// SIMATIC S7-200 project (STEP 7-Micro/WIN), CPU 226 CN REL 02.01

ORGANIZATION_BLOCK MAIN:OB1
TITLE=PROGRAM COMMENTS
BEGIN
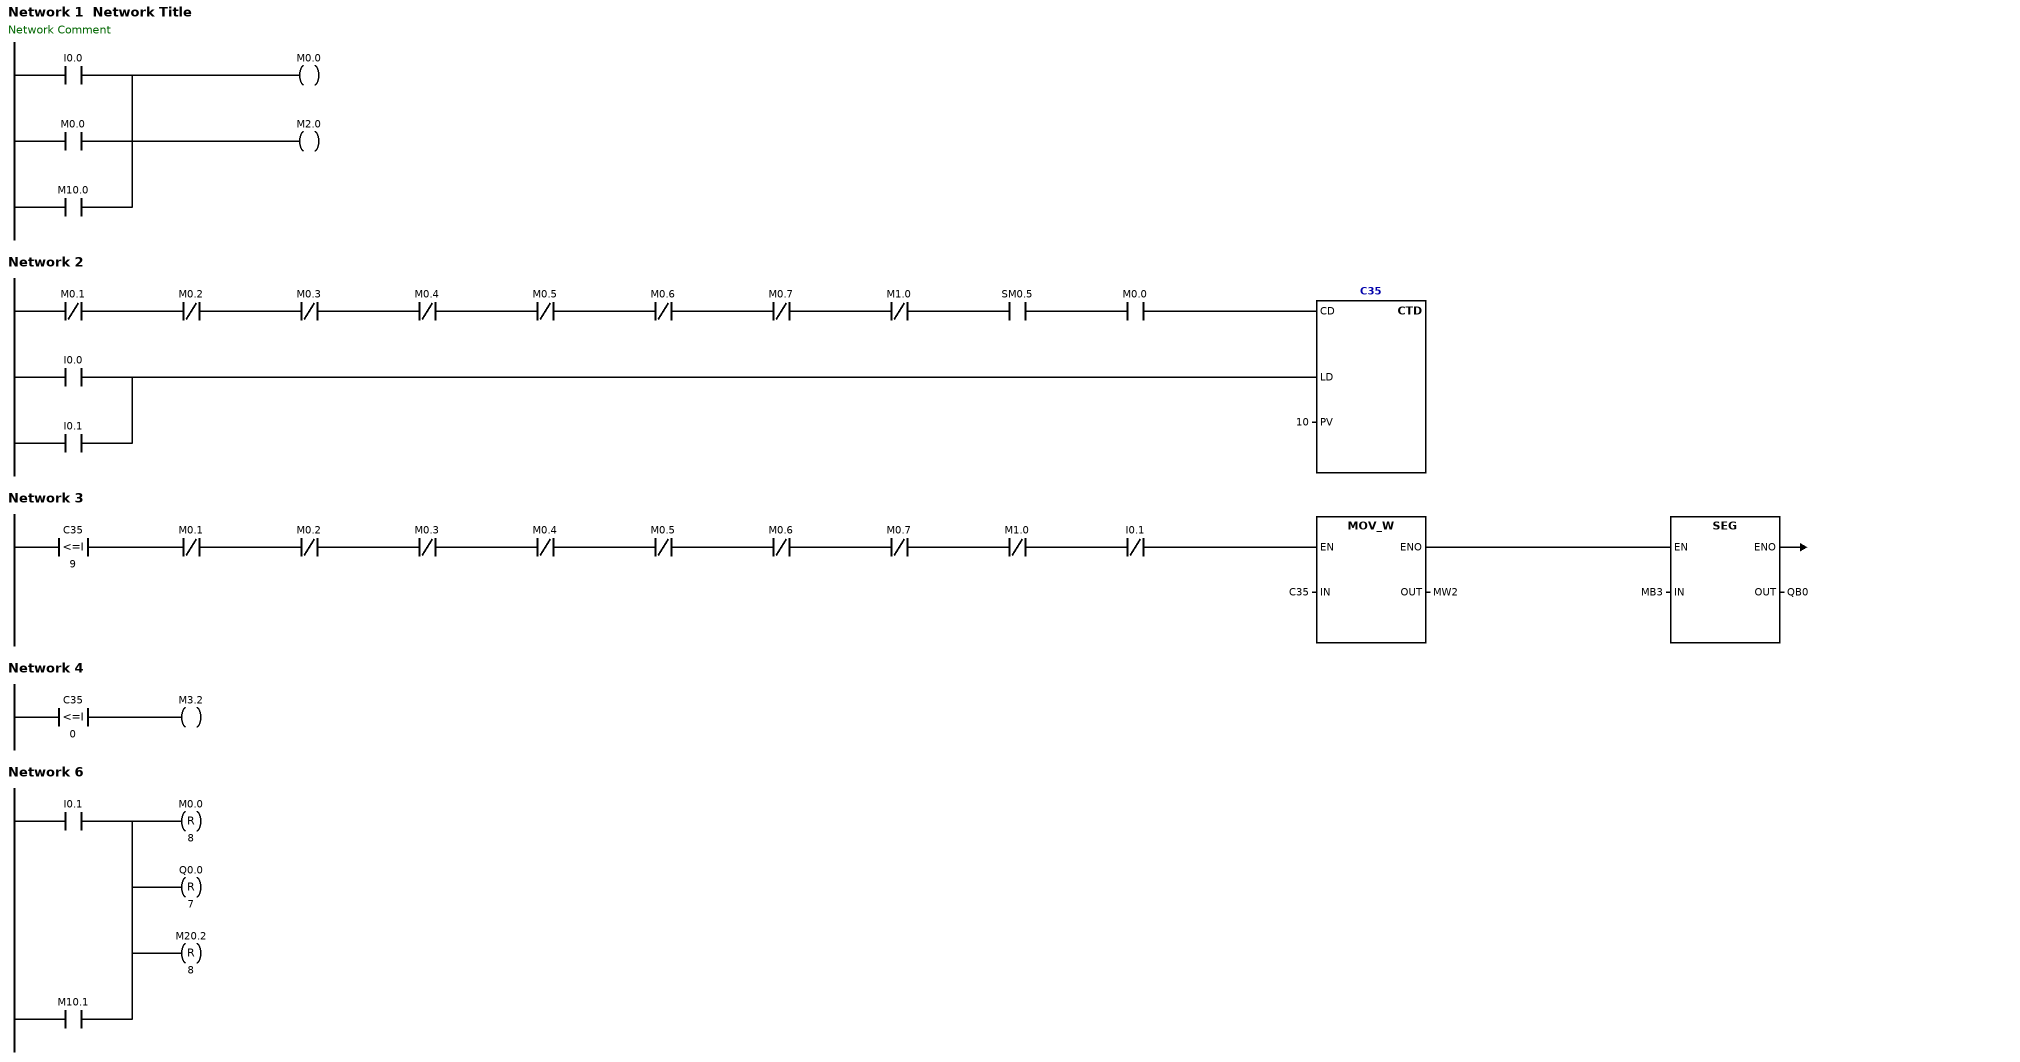
Network 1 // Network Title
// Network Comment
// (network saved uncompiled; LAD cells follow)
// row 0: c0 -| |- I0.0 v  c1 --  c2 -( ) M0.0
// row 1: c0 -| |- M0.0 ^v  c1 --  c2 -( ) M2.0
// row 2: c0 -| |- M10.0 ^
Network 2
LDN    M0.1
AN     M0.2
AN     M0.3
AN     M0.4
AN     M0.5
AN     M0.6
AN     M0.7
AN     M1.0
A      SM0.5
A      M0.0
LD     I0.0
O      I0.1
CTD    C35, 10
Network 3
LDW<=  C35, 9
AN     M0.1
AN     M0.2
AN     M0.3
AN     M0.4
AN     M0.5
AN     M0.6
AN     M0.7
AN     M1.0
AN     I0.1
MOVW   C35, MW2
AENO
SEG    MB3, QB0
Network 4
LDW<=  C35, 0
=      M3.2
Network 6
// (network saved uncompiled; LAD cells follow)
// row 0: c0 -| |- I0.1 v  c1 -(R) M0.0, 8
// row 1: c0 ^v  c1 -(R) Q0.0, 7
// row 2: c0 ^v  c1 -(R) M20.2, 8
// row 3: c0 -| |- M10.1 ^
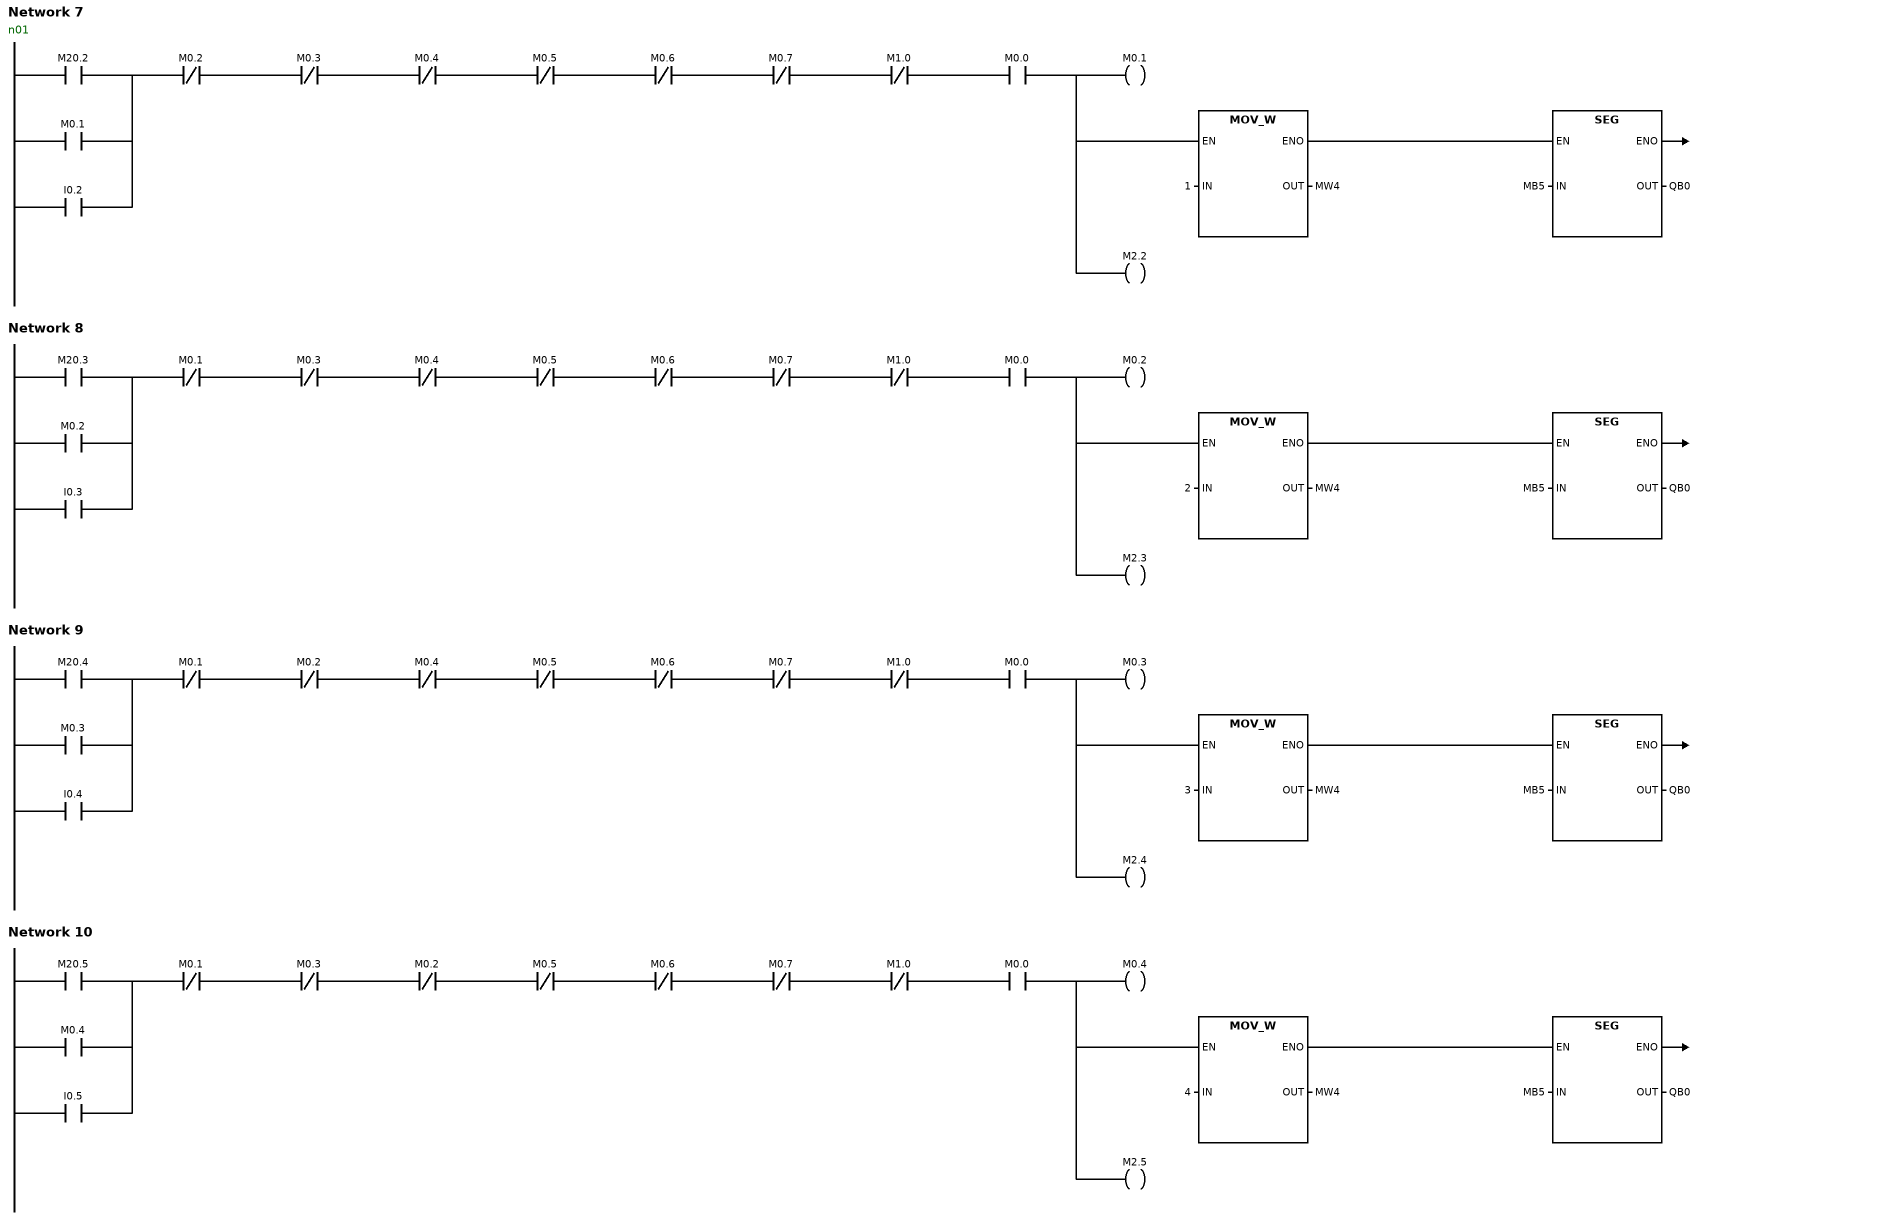
Network 7
// n01
LD     M20.2
O      M0.1
O      I0.2
AN     M0.2
AN     M0.3
AN     M0.4
AN     M0.5
AN     M0.6
AN     M0.7
AN     M1.0
A      M0.0
LPS
=      M0.1
MOVW   1, MW4
AENO
SEG    MB5, QB0
LPP
=      M2.2
Network 8
LD     M20.3
O      M0.2
O      I0.3
AN     M0.1
AN     M0.3
AN     M0.4
AN     M0.5
AN     M0.6
AN     M0.7
AN     M1.0
A      M0.0
LPS
=      M0.2
MOVW   2, MW4
AENO
SEG    MB5, QB0
LPP
=      M2.3
Network 9
LD     M20.4
O      M0.3
O      I0.4
AN     M0.1
AN     M0.2
AN     M0.4
AN     M0.5
AN     M0.6
AN     M0.7
AN     M1.0
A      M0.0
LPS
=      M0.3
MOVW   3, MW4
AENO
SEG    MB5, QB0
LPP
=      M2.4
Network 10
LD     M20.5
O      M0.4
O      I0.5
AN     M0.1
AN     M0.3
AN     M0.2
AN     M0.5
AN     M0.6
AN     M0.7
AN     M1.0
A      M0.0
LPS
=      M0.4
MOVW   4, MW4
AENO
SEG    MB5, QB0
LPP
=      M2.5
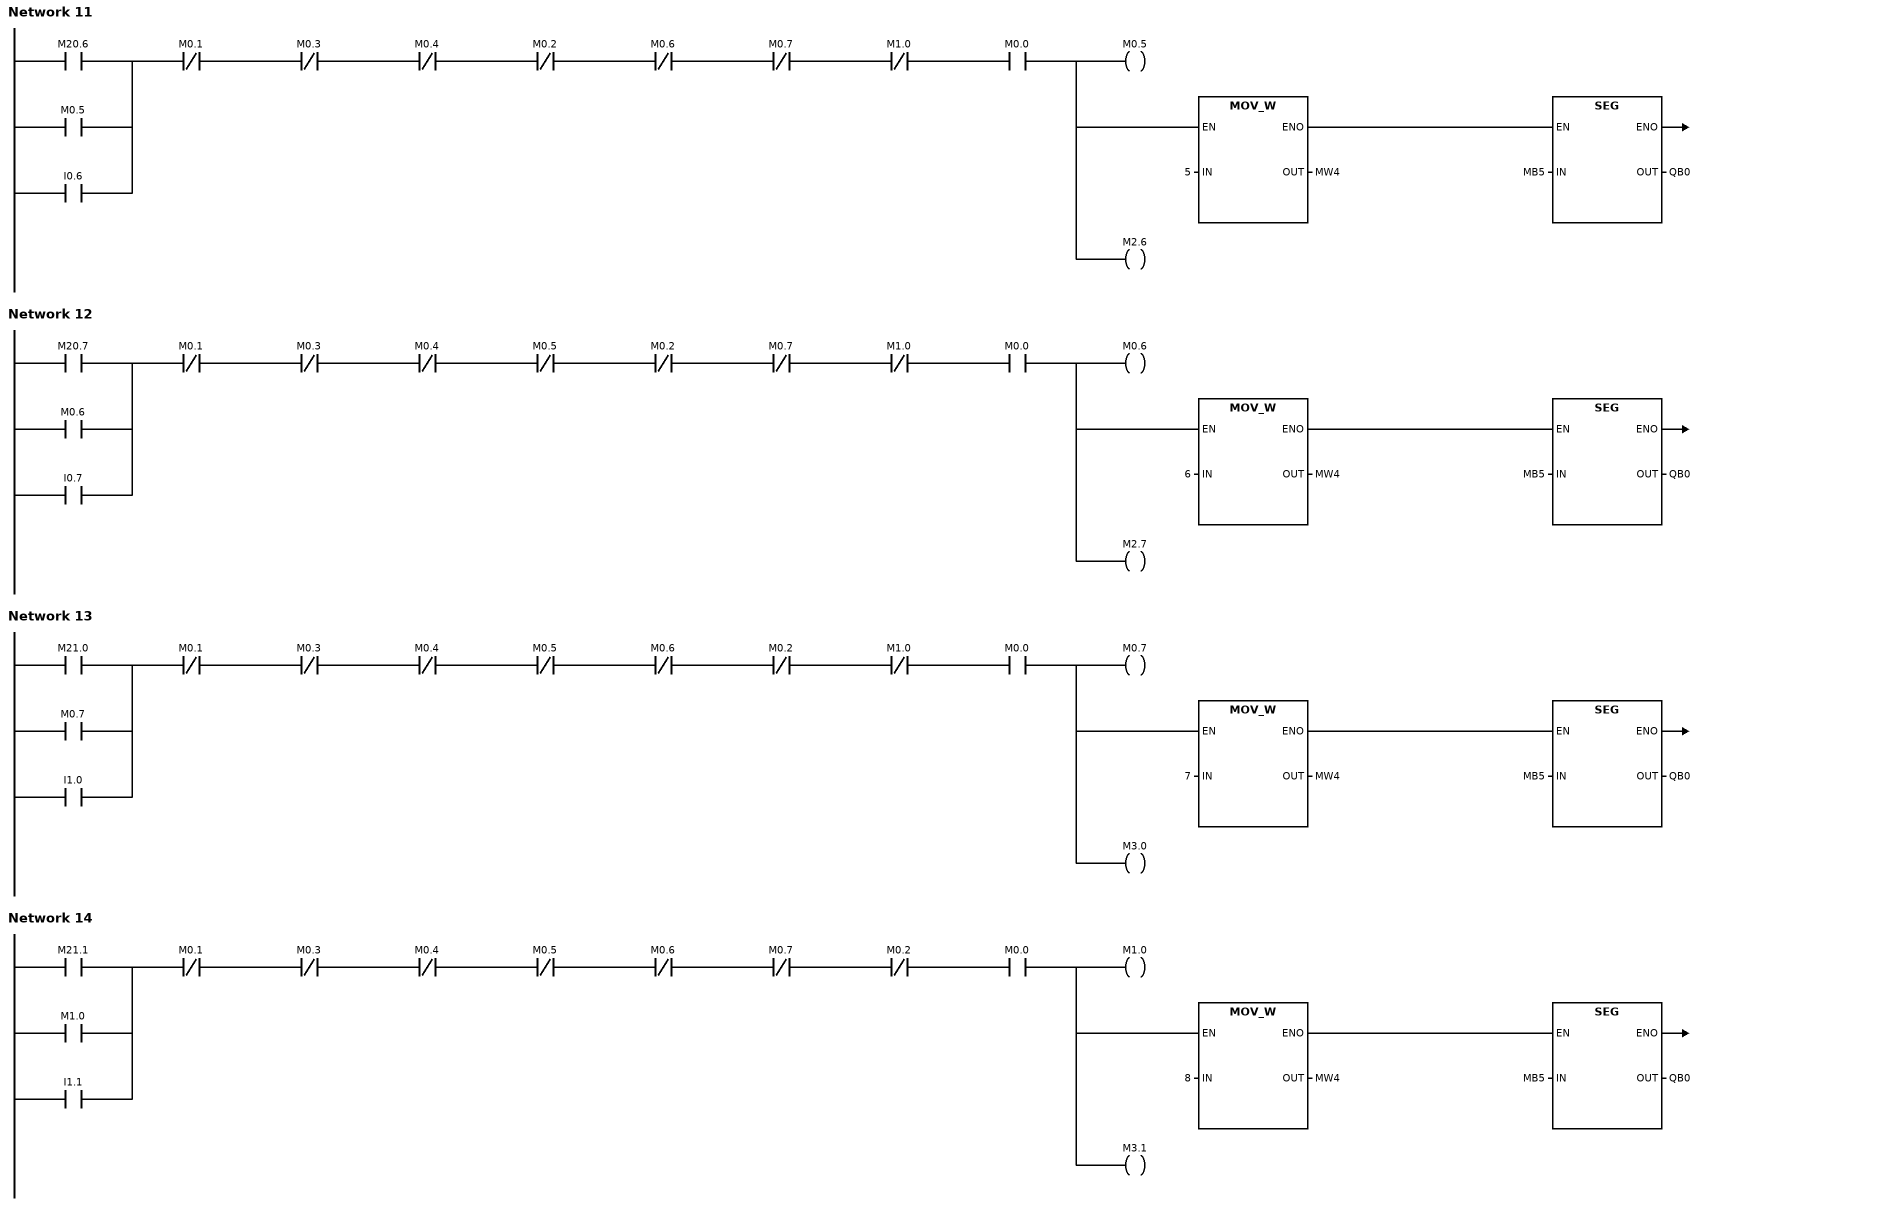
Network 11
LD     M20.6
O      M0.5
O      I0.6
AN     M0.1
AN     M0.3
AN     M0.4
AN     M0.2
AN     M0.6
AN     M0.7
AN     M1.0
A      M0.0
LPS
=      M0.5
MOVW   5, MW4
AENO
SEG    MB5, QB0
LPP
=      M2.6
Network 12
LD     M20.7
O      M0.6
O      I0.7
AN     M0.1
AN     M0.3
AN     M0.4
AN     M0.5
AN     M0.2
AN     M0.7
AN     M1.0
A      M0.0
LPS
=      M0.6
MOVW   6, MW4
AENO
SEG    MB5, QB0
LPP
=      M2.7
Network 13
LD     M21.0
O      M0.7
O      I1.0
AN     M0.1
AN     M0.3
AN     M0.4
AN     M0.5
AN     M0.6
AN     M0.2
AN     M1.0
A      M0.0
LPS
=      M0.7
MOVW   7, MW4
AENO
SEG    MB5, QB0
LPP
=      M3.0
Network 14
LD     M21.1
O      M1.0
O      I1.1
AN     M0.1
AN     M0.3
AN     M0.4
AN     M0.5
AN     M0.6
AN     M0.7
AN     M0.2
A      M0.0
LPS
=      M1.0
MOVW   8, MW4
AENO
SEG    MB5, QB0
LPP
=      M3.1
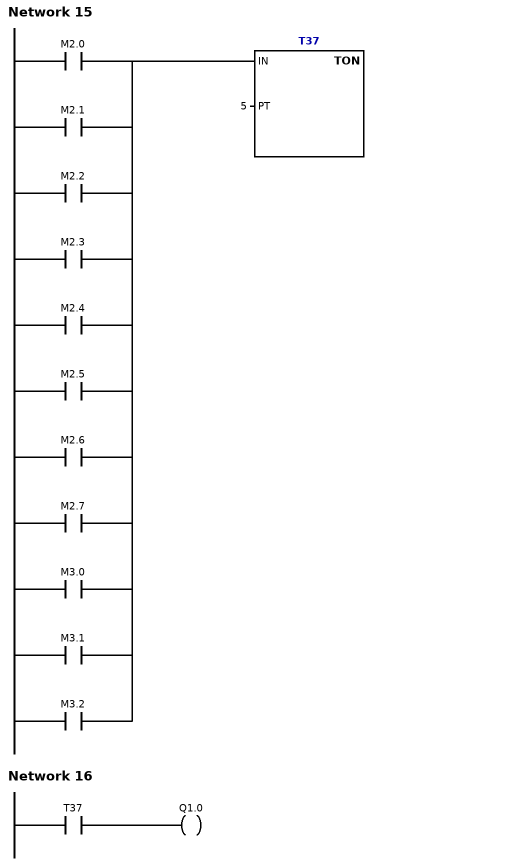
Network 15
LD     M2.0
O      M2.1
O      M2.2
O      M2.3
O      M2.4
O      M2.5
O      M2.6
O      M2.7
O      M3.0
O      M3.1
O      M3.2
TON    T37, 5
Network 16
LD     T37
=      Q1.0
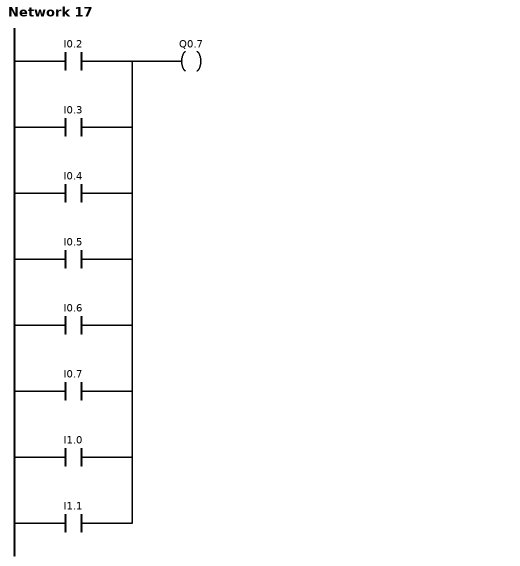
Network 17
LD     I0.2
O      I0.3
O      I0.4
O      I0.5
O      I0.6
O      I0.7
O      I1.0
O      I1.1
=      Q0.7
END_ORGANIZATION_BLOCK
